// Mitsubishi GX Works2 project: 拨片式分拣两段皮带   PLC: FX2N/FX2NC

PROGRAM MAIN
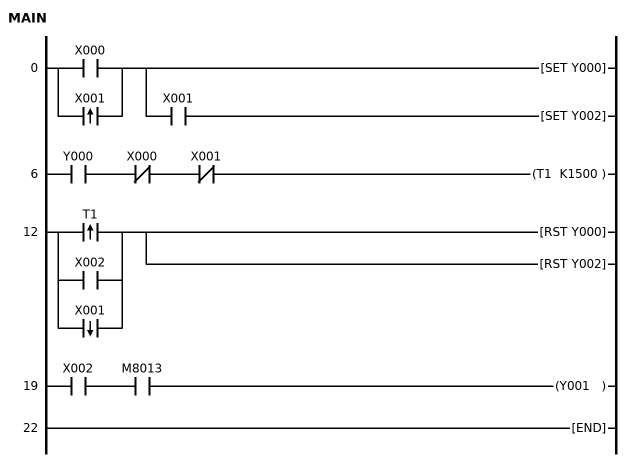
0     LD      X000
      ORP     X001
      SET     Y000
      AND     X001
      SET     Y002
6     LD      Y000
      ANI     X000
      ANI     X001
      OUT     T1 K1500
12    LDP     T1
      OR      X002
      ORF     X001
      RST     Y000
      RST     Y002
19    LD      X002
      AND     M8013
      OUT     Y001
22    END
END_PROGRAM
